// TwinCAT 3 PLC project PlcTc3JsonXmlSampleJsonDomReader
// ProgramVersion: 3.1.4021.2
// libraries:
//   Tc2_Standard, * (Beckhoff Automation GmbH)
//   Tc2_System, * (Beckhoff Automation GmbH)
//   Tc3_JsonXml, * (Beckhoff Automation GmbH)
//   Tc3_Module, * (Beckhoff Automation GmbH)
// project tree:
//   DUTs/ ST_ReceivedData.TcDUT
//   / PlcTask.TcTTO
//   POUs/ MAIN.TcPOU
// real-time tasks:
//   TASK PlcTask: cycle T#10ms, priority 20, ADS port 350

CONFIGURATION PlcTc3JsonXmlSampleJsonDomReader
    RESOURCE PLC ON TwinCAT3
        TASK PlcTask(INTERVAL := T#10ms, PRIORITY := 20);
        PROGRAM MAIN WITH PlcTask : MAIN;
    END_RESOURCE
END_CONFIGURATION

// ---- DUTs/ST_ReceivedData.TcDUT
TYPE ST_ReceivedData :
STRUCT
	serialNumber 	: STRING(255);
	batteryVoltage 	: STRING(255);
	clickType		: STRING(255);
END_STRUCT
END_TYPE

// ---- POUs/MAIN.TcPOU
PROGRAM MAIN
VAR
	(* JSON *)
	fbJson 			: FB_JsonDomParser;
	jsonDoc 		: SJsonValue;
	jsonProp		: SJsonValue;
	jsonValue		: SJsonValue;
	bHasMember		: BOOL;
  	sMessage 		: STRING(255) := '{"serialNumber":"G030PT028191AC4R","batteryVoltage":"1547mV","clickType":"SINGLE"}';
	stReceivedData	: ST_ReceivedData;
END_VAR

(* Retrieve JSON content *)
jsonDoc := fbJson.ParseDocument(sMessage);
bHasMember := fbJson.HasMember(jsonDoc, 'serialNumber');
IF (bHasMember) THEN
	  bHasMember := FALSE;
	  jsonProp := fbJson.FindMember(jsonDoc, 'serialNumber');
	  stReceivedData.serialNumber := fbJson.GetString(jsonProp);
END_IF

bHasMember := fbJson.HasMember(jsonDoc, 'batteryVoltage');
IF (bHasMember) THEN
	  bHasMember := FALSE;
	  jsonProp := fbJson.FindMember(jsonDoc, 'batteryVoltage');
	  stReceivedData.batteryVoltage := fbJson.GetString(jsonProp);
END_IF		

bHasMember := fbJson.HasMember(jsonDoc, 'clickType');
IF (bHasMember) THEN
	  bHasMember := FALSE;
	  jsonProp := fbJson.FindMember(jsonDoc, 'clickType');
	  stReceivedData.clickType := fbJson.GetString(jsonProp);
END_IF

END_PROGRAM
